Staubli VAL3: trigger.pgx

public program trigger(num handle_, bool& result_[])
begin
  // trigger image acquire and evaluation
  //call sendCommand(handle_,"sw8",result_)
  call setEventAndWait(handle_,8,result_)
end
